// TIA Portal V19 export
DATA_BLOCK "Projekt_2B_Robotgrinder_DB"   // DB1
// stored: InstanceOfName Projekt_2B_Robotgrinder, InstanceOfType FB
"Projekt_2B_Robotgrinder"
BEGIN
END_DATA_BLOCK
